PROGRAM MAIN
VAR	

	FB_EdgeDetector	: fb_EdgeDetector;
	bTaster 		: BOOL;
	bLampe			: BOOL;
	timeDelay		: TIME := T#200MS;
	bDummy			: BOOL;

END_VAR

FB_EdgeDetector(bSignal := bTaster, timeON := timeDelay, bRisingEdge =>bLampe);
IF bLampe THEN
	bDummy := TRUE;
ELSE
	bDummy := FALSE;
END_IF

END_PROGRAM

(* stored: Version 1.1.0.1, ProductVersion 3.1.4024.12
   POU MAIN: Id {3b07cc55-1f68-4919-a9db-3257e04150e1}, SpecialFunc None *)
